(* PLC project Water Tower, Blank VGP 1.0 *)
(* stored: creationDateTime 2016-05-18T21:14:07, modificationDateTime 2020-01-10T16:41:08 *)

PROGRAM My_Program
  VAR
    temp AT %IW0 : INT;
    temp_filtered AT %QW6 : INT;
    Alarm AT %QX0.5 : BOOL;
    min_sp AT %QW1 : INT := 18333;
    max_sp AT %QW2 : INT := 23889;
    mode_register AT %QW3 : INT := 2;
    heat_register AT %QW4 : INT := 1;
    cool_register AT %QW5 : INT;
    heat AT %QX0.0 : BOOL;
    cool AT %QX0.1 : BOOL;
    heat_man AT %QX1.0 : BOOL;
    heat_auto AT %QX1.1 : BOOL;
    cool_man AT %QX1.2 : BOOL;
    cool_auto AT %QX1.3 : BOOL;
  END_VAR
  VAR  (* added by the conversion: wires and edge detectors of the diagram *)
    _EQ1_OUT : BOOL;
  END_VAR

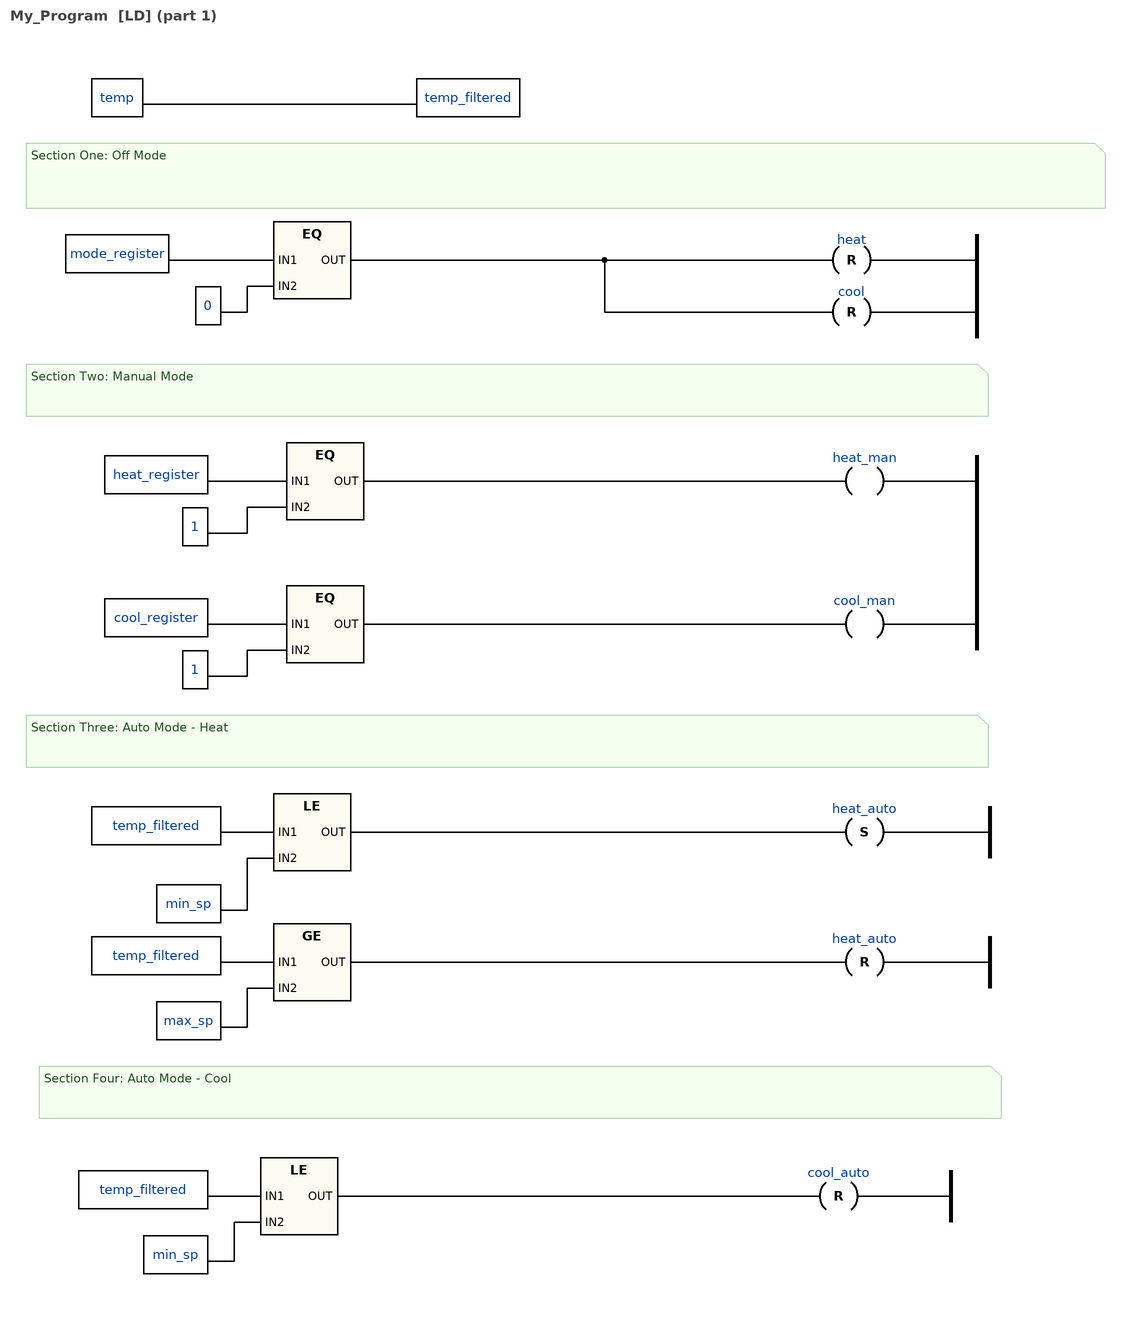
(* LD diagram, written out as Structured Text *)
temp_filtered := temp;
(* Section One: Off Mode *)
_EQ1_OUT := mode_register = 0;
IF _EQ1_OUT THEN heat := FALSE; END_IF;
IF _EQ1_OUT THEN cool := FALSE; END_IF;
(* Section Two: Manual Mode *)
heat_man := heat_register = 1;
cool_man := cool_register = 1;
(* Section Three: Auto Mode - Heat *)
IF temp_filtered <= min_sp THEN heat_auto := TRUE; END_IF;
IF temp_filtered >= max_sp THEN heat_auto := FALSE; END_IF;
(* Section Four: Auto Mode - Cool *)
IF temp_filtered <= min_sp THEN cool_auto := FALSE; END_IF;
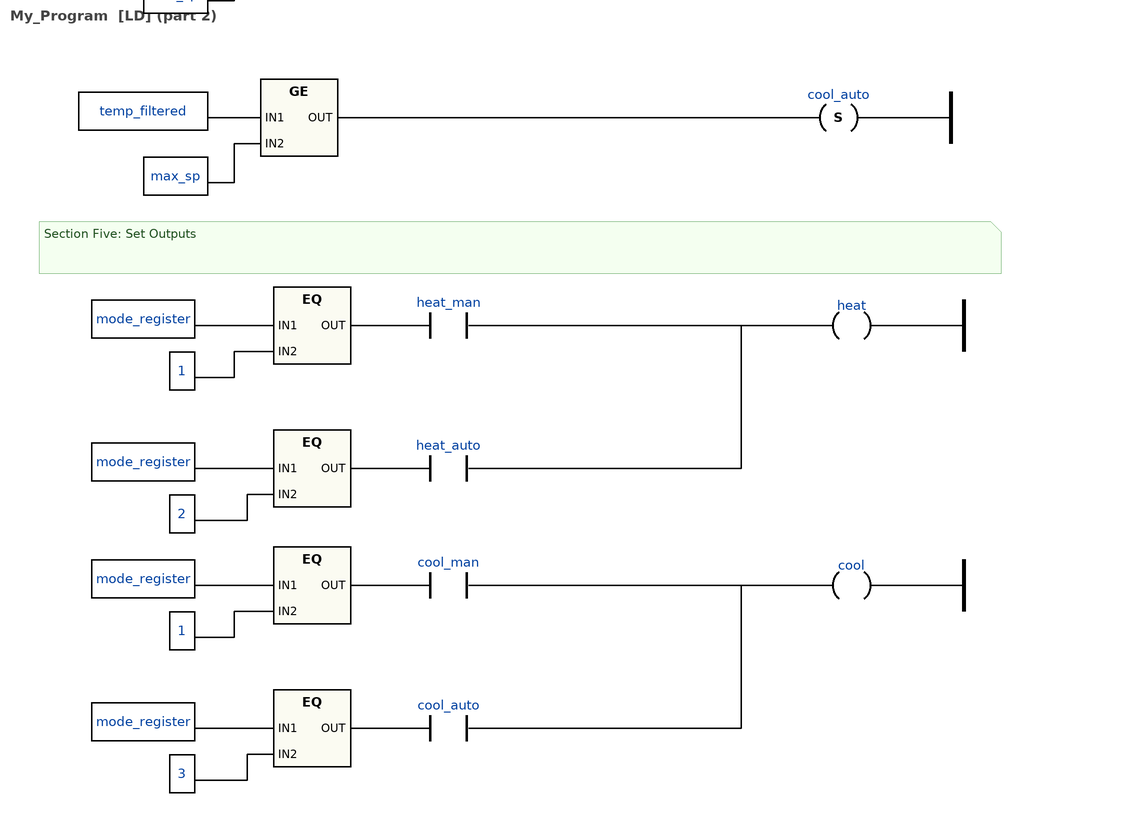
IF temp_filtered >= max_sp THEN cool_auto := TRUE; END_IF;
(* Section Five: Set Outputs *)
heat := mode_register = 1 AND heat_man OR mode_register = 2 AND heat_auto;
cool := mode_register = 1 AND cool_man OR mode_register = 3 AND cool_auto;
END_PROGRAM

FUNCTION_BLOCK Level_Filtering
  VAR_INPUT
    raw_level : INT;
  END_VAR
  VAR
    level_real : REAL;
    avg : LREAL;
    level_array : ARRAY[1..20] OF REAL;
    i : INT;
    current_array_pos : INT := 1;
  END_VAR
  VAR_OUTPUT
    filtered_level : INT;
  END_VAR

            (* Level Conversion *)
level_real := INT_TO_REAL(raw_level);
level_real := level_real - 107.0;
level_real := level_real * 0.483091;
level_real := level_real * 100.0;

(* Store value in average array *)
level_array[current_array_pos] := level_real;
current_array_pos := current_array_pos + 1;

(* Prevent array_pos overflow *)
if current_array_pos > 20 then
  current_array_pos := 1;
end_if;

(* Calculate average *)
avg := 0.0;
i := 1;
while (i < 21) do
  avg := avg + REAL_TO_LREAL(level_array[i]);
  i := i + 1;
end_while;
avg := avg / 20.0;

(* Set output value *)
filtered_level := LREAL_TO_INT(avg);
          
END_FUNCTION_BLOCK

CONFIGURATION Config0
  RESOURCE Res0 ON PLC
    TASK TaskMain(INTERVAL := T#50ms, PRIORITY := 0);
    PROGRAM Inst0 WITH TaskMain : My_Program;
  END_RESOURCE
END_CONFIGURATION
